# EPICS autosave request: BPMApp/Db/BPMFmc130m_4ch_settings.req
$(P)$(R)ADCRandEn
$(P)$(R)ADCDithEn
$(P)$(R)ADCShdnEn
$(P)$(R)ADCPgaEn
